PROGRAM POU
VAR
	xCordinates :  ARRAY[0..10000] OF INT;
	yCordinates :  ARRAY[0..10000] OF INT;
	mcPower : MC_Power;
	mcSetPosition: MC_SetPosition;
	mcMoveAboslute: MC_MoveAbsolute;
	mcMoveRelative: MC_MoveRelative;
	mcMoveVelocity: MC_MoveVelocity;
	mcReset:MC_Reset;
	mcHalt:MC_Halt;
	mcStop:MC_Stop;
	
	bEnable : BOOL;
	bExecute_SPOS :BOOL;
	bExecute_MABS :BOOL;
	bExecute_MREL :BOOL;
	bExecute_RES :BOOL;
	bExecute_VEL :BOOL;
	bExecute_HALT :BOOL;
	bExecute_STOP :BOOL;
	
	fVelocity:LREAL;
	fPosition:LREAL;
	fAccel:LREAL;
END_VAR

mcPower.Enable:=true;

END_PROGRAM

(* stored: Version 1.1.0.1, ProductVersion 3.1.4024.12
   POU POU: Id {a67fbdca-72a1-41f4-92e4-b24578acb3c9}, SpecialFunc None *)
